Yaskawa INFORM job: _DEL23.JBI

/JOB
//NAME _DEL23
//POS
///NPOS 0,0,0,0,0,0
//INST
///DATE 2018/08/30 11:48
///ATTR SC,RW,SY
///GROUP1 ST1
///LVARS 5,0,5,0,0,0,0,0
NOP
END
